FUNCTION_BLOCK fb_ele_reset
VAR_IN_OUT
	var_ref_ele : ref_ele_io;
END_VAR
VAR_INPUT
	in_flg_reset : BOOL;
END_VAR
VAR_OUTPUT
	out_flg_resetDone : bool;
END_VAR
VAR
	var_process: INT;
	fbi_ton1: TON;
END_VAR


fbi_ton1(IN:= , PT:=T#100MS , Q=> , ET=> );
IF NOT in_flg_reset THEN
	var_process := 0;
	out_flg_resetDone := FALSE;
	var_ref_ele.output.out_flg_reset := FALSE;
END_IF
CASE var_process OF
	0:
		IF in_flg_reset THEN
			fbi_ton1.IN := FALSE;
			var_process := 1;
		END_IF
	1:
		var_ref_ele.output.out_flg_eleA := FALSE;
		var_ref_ele.output.out_flg_eleB := FALSE;
		var_ref_ele.output.out_flg_reset := TRUE;
		var_ref_ele.param.var_mutex := 0;
		fbi_ton1.IN := TRUE;
		IF fbi_ton1.Q THEN
			var_process := 2;
		END_IF
	2:
		var_ref_ele.output.out_flg_reset := FALSE;
		out_flg_resetDone := TRUE;
		var_process := 3;
	3:
		out_flg_resetDone := FALSE;
END_CASE

END_FUNCTION_BLOCK

(* stored: Version 1.1.0.1, ProductVersion 3.1.4024.11
   POU fb_ele_reset: Id {a3abecf7-2748-4542-b61b-26de034d24d8}, SpecialFunc None *)
